Staubli VAL3: OnF3.pgx

program OnF3()
begin
  //删除
  call Delete()
end
